FUNCTION_BLOCK FB_KOH

VAR_INPUT
	bEnableKOHFunction				: BOOL; // Aktiverar KOH via driftindikering av VS-pump
	bBlockKOHFunction				: BOOL; // Blockera KOH via annan källa		
	bExceptionKOH					: BOOL; // Aktiverar undantags-funktion		
    wMondayOn						: WORD; // Tillslagstid för måndag [0000-2400]
    wMondayOff						: WORD; // Frånslagstid för måndag [0000-2400]
    wTuesdayOn						: WORD; // Tillslagstid för tisdag [0000-2400]
    wTuesdayOff						: WORD; // Frånslagstid för tisdag [0000-2400]
    wWednesdayOn					: WORD; // Tillslagstid för onsdag [0000-2400]
    wWednesdayOff					: WORD; // Frånslagstid för onsdag [0000-2400]
    wThursdayOn						: WORD; // Tillslagstid för torsdag [0000-2400]
    wThursdayOff					: WORD; // Frånslagstid för torsdag [0000-2400]
    wFridayOn						: WORD; // Tillslagstid för fredag [0000-2400]
    wFridayOff						: WORD; // Frånslagstid för fredag [0000-2400]
    wSaturdayOn						: WORD; // Tillslagstid för lördag [0000-2400]
    wSaturdayOff					: WORD; // Frånslagstid för lördag [0000-2400]
    wSundayOn						: WORD; // Tillslagstid för söndag [0000-2400]
    wSundayOff						: WORD; // Frånslagstid för söndag [0000-2400]
	
	diSystemCalcSetpoint			: DINT; // Systemets aktuella beräknade börvärde [0000-2400]
	diDownRampTime					: DINT; // Upprampning av förskjutning tillbaka till ursprungsberäkning av börvärde [0-1000 minuter (0-100)]
	diSPEveningReduction			: DINT; // Inställning börvärdessänka kvällstid måndag-söndag [0-1000 (0-100°C)]
	diSPWeekendReduction			: DINT; // Inställning börvärdessänka helgtid [0-1000 (0-100°C)]
	diSPHolidayReduction			: DINT; // Inställning börvärdessänka helgdagar [0-1000 (0-100°C)]
	diSPExceptionReduction			: DINT; // Inställning börvärdessänka undantagssänka [0-1000 (0-100°C)]
	diActualAverageRoomTemp			: DINT; // Aktuellt medelvärde rumstemperatur
	diAllowedMinRoomTemp			: DINT; // Lägsta tillåtna rumsmedeltemperatur [0-1000 (0-100°C)]
END_VAR

VAR_OUTPUT	
	bKOHActive						: BOOL; // KOH-funktion aktiv
	bKOHBlocked						: BOOL; // KOH-funktion blockerad från annan källa
	bAlarmBlocked					: BOOL; // Alarm, KOH-funktion blockerad [B]
	bAlarmMinTemp					: BOOL; // Lägsta rumstemperaturen uppnådd [B]
	diKOHCalcOffset					: DINT; // Aktuellt nytt beräknat börvärde
	bRampTimeActive					: BOOL; // Ramp-funktion aktiv
END_VAR

VAR
// Sytemtid	
	fbSystemTime 					: FB_SystemTime;
// Funktionsblock
	fbTidkanalKOH					: FB_TidKanalDrift; // Tidkanalsblock
	fbSwedishHolidays				: FB_SwedishHolidays; // Block för beräkning av svenska helgdagar
	fbRamp							: FB_Ramp; // Rampblock
	fbSel							: FB_Sel; // Selectblock av korrekt förskjutning
	fbPIDCascade					: FB_PID; // PID för kaskad av förskjutning

// Lokala variabler	
	bVarTidKanalAktiv				: BOOL; // Lokal variabel, tidkanal för drift aktiv
	dActDate						: DATE_AND_TIME; 	
	dtVarSystemTime 				: DATE_AND_TIME;
	todVarTimeOfDay					: TIME_OF_DAY;
	dDate 							: DATE; // Aktuellt datum
	todActTime						: TIME_OF_DAY; // Aktuellt klockslag
	iVarActDay						: INT; // Lokal variabel, aktuell dag. Måndag=1, Tisdag=2, Onsdag=3, Torsdag=4, Fredag=5, Lördag=6, Söndag=0
	bVarVardagAct					: BOOL; // Lokal variabel, Måndag-fredag aktiv
	bVarVeckoslutAct				: BOOL; // Lokal variabel, vanlig lördag-söndag aktiv
	bVarHelgdagAktiv				: BOOL; // Lokal variabel, någon helgdag är aktiv
	bVarExceptionAct				: BOOL; // Lokal variabel, undantagssänka aktiv
	
	bVarTKVardagAct					: BOOL; // Lokal variabel, Måndag-fredag aktiv
	bVarTKVeckoslutAct				: BOOL; // Lokal variabel, vanlig lördag-söndag aktiv
	bVarTKExceptionAct				: BOOL; // Lokal variabel, undantagssänka aktiv
	
	diVarSelOutPut					: DINT; // Lokal variabel, temp-värde
	diVarOffsetValue				: DINT; // Lokal variabel, värde som ska förskjuta beräknat börvärde
END_VAR

fbSystemTime();
dtVarSystemTime:= 	fbSystemTime.dtSystemTime;
todActTime:= 		todVarTimeOfDay;
dDate:= 			TO_DATE(dtVarSystemTime);
todVarTimeOfDay:= 	TO_TOD (fbSystemTime.dtSystemTime); 
// Kör hela KOH om det inte är blockerat
IF NOT bBlockKOHFunction THEN

//===========Startar KOH om pumpen för värmesystemet är i drift===========//
IF bEnableKOHFunction THEN

//===========Block för att beräkna svenska helgdagar===========//	
fbSwedishHolidays();

//===========Tidkanal för aktivering av KOH===========//
fbTidkanalKOH(
	bEn:= 						,
	wMondayOn:= 				wMondayOn,
	wMondayOff:= 				wMondayOff,
	wTuesdayOn:= 				wTuesdayOn,
	wTuesdayOff:= 				wTuesdayOff,
	wWednesdayOn:= 				wWednesdayOn,
	wWednesdayOff:= 			wWednesdayOff,
	wThursdayOn:= 				wThursdayOn,
	wThursdayOff:= 				wThursdayOff,
	wFridayOn:= 				wFridayOn,
	wFridayOff:= 				wFridayOff,
	wSaturdayOn:= 				wSaturdayOn,
	wSaturdayOff:= 				wSaturdayOff,
	wSundayOn:= 				wSundayOn,
	wSundayOff:= 				wSundayOff,
	bOn=> 						bVarTidKanalAktiv);
	
//=========== Aktiverar mån-fre, lör-sön, helgdag, undantag i fallande prio===========//
// Beräknar dag 0-6 
iVarActDay:=fc_Day_Of_Year(IDATE:=TO_DATE (dDate));
// Beräknar mån-fre 1-5
IF (iVarActDay >0 AND iVarActDay <5) AND NOT bVarHelgdagAktiv THEN
	bVarVardagAct:= TRUE;	
// Beräknar lör-sön 6,0
ELSIF (iVarActDay = 7 OR iVarActDay = 0) AND NOT bVarHelgdagAktiv THEN
	bVarVardagAct	:= FALSE;	
	bVarVeckoslutAct:= TRUE;
	bVarHelgdagAktiv:= FALSE;
	bVarExceptionAct:= FALSE;	
// Beräknar helgdag
ELSIF fbSwedishHolidays.bHelgDagAktiv THEN
	bVarVardagAct	:= FALSE;	
	bVarVeckoslutAct:= FALSE;
	bVarHelgdagAktiv:= TRUE;
	bVarExceptionAct:= FALSE;
// Beräknar undantag
ELSIF bExceptionKOH THEN
	bVarVardagAct	:= FALSE;	
	bVarVeckoslutAct:= FALSE;
	bVarHelgdagAktiv:= FALSE;
	bVarExceptionAct:= TRUE;
ELSE
	bVarVardagAct	:= FALSE;	
	bVarVeckoslutAct:= FALSE;
	bVarHelgdagAktiv:= FALSE;
	bVarExceptionAct:= FALSE;
END_IF


// Startar KOH via tidkanal och aktuellt veckoläge
IF bVarTidKanalAktiv AND bVarVardagAct THEN
	bVarTKVardagAct:=	 	TRUE;
	bVarTKVeckoslutAct:= 	FALSE;
	bVarHelgdagAktiv:=	 	FALSE;
	bVarTKExceptionAct:= 	FALSE;
ELSIF bVarTidKanalAktiv AND bVarVeckoslutAct THEN	
	bVarTKVardagAct:= 		FALSE;
	bVarTKVeckoslutAct:= 	TRUE;
	bVarHelgdagAktiv:= 		FALSE;
	bVarTKExceptionAct:= 	FALSE;
ELSIF bVarTidKanalAktiv AND bVarHelgdagAktiv THEN	
	bVarTKVardagAct:= 		FALSE;
	bVarTKVeckoslutAct:= 	FALSE;
	bVarHelgdagAktiv:= 		TRUE;
	bVarTKExceptionAct:= 	FALSE;
ELSIF bVarExceptionAct THEN	
	bVarTKVardagAct:= 		FALSE;
	bVarTKVeckoslutAct:= 	FALSE;
	bVarHelgdagAktiv:= 		FALSE;
	bVarTKExceptionAct:=	TRUE;
END_IF

IF bVarTKVardagAct OR bVarTKVeckoslutAct OR bVarHelgdagAktiv OR bVarTKExceptionAct THEN
// Väljer korrekt offset i fallande prio om någon förskjutning ska ske
fbSel(
	diSelVal01:= 		diSPEveningReduction, 
	diSelVal02:= 		diSPWeekendReduction, 
	diSelVal03:= 		diSPHolidayReduction, 
	diSelVal04:= 		diSPExceptionReduction, 
	bEnabelVal01:= 		bVarTKVardagAct, 
	bEnabelVal02:= 		bVarTKVeckoslutAct, 
	bEnabelVal03:= 		bVarHelgdagAktiv, 
	bEnabelVal04:= 		bVarTKExceptionAct, 
	diOutPut=> 			diVarSelOutPut);
ELSE diVarSelOutPut:= 0;
	
END_IF

// Kör valt värde genom nedrampning
fbRamp(
	diInPutValue:= 		diVarSelOutPut, 
	diRampUpTime:= 		0, 
	diRampDownTime:= 	diDownRampTime, 
	diOutPutValue=> 	diVarOffsetValue, 
	bActive=> 			bRampTimeActive, 
	bUpDown=> 			);

// Larm för låg rumstemperatur	
IF diActualAverageRoomTemp <= diAllowedMinRoomTemp THEN
	bAlarmMinTemp:= TRUE; ELSE	
	bAlarmMinTemp:= FALSE;
END_IF

// PID som rampar ner förskjutning vid "kallt" i rum
fbPIDCascade(
	bEn:= 				bVarTKVardagAct OR bVarTKVeckoslutAct OR bVarHelgdagAktiv OR bVarTKExceptionAct,
	nPV:= 				diActualAverageRoomTemp,
	nSP:= 				diAllowedMinRoomTemp, 
	nP:= 				, 
	nI:= 				, 
	nD:= 				, 
	nDF:= 				, 
	nMAX:= 				diVarOffsetValue,
	nMIN:= 				0,
	nInitValue:= 		,
	nDeactValue:= 		diVarOffsetValue,
	bInvert:= 			,
	nY=> 				);


diKOHCalcOffset:= (diSystemCalcSetpoint - (diVarOffsetValue - fbPIDCascade.nY));




END_IF

END_IF
bAlarmBlocked:= 	bBlockKOHFunction;
bKOHBlocked:= 		bBlockKOHFunction;
diKOHCalcOffset:= 	diSystemCalcSetpoint;

END_FUNCTION_BLOCK

(* stored: Version 1.1.0.1, ProductVersion 3.1.4024.11
   POU FB_KOH: Id {0498d426-6b37-4146-a330-619b12b2afd4}, SpecialFunc None *)
